// TIA Portal V18 export
TYPE "LGasp_typeRigaProdfromPC"
// stored: IsFailsafeCompliant false
   STRUCT
      piecestodo : DInt;   // Pezzi da fare
      ID : DInt;   // ID riga di produzione
      tipoarticolo : DInt;   // tipo articolo
      info : Struct   // info varie variabili da macchina a macchina
         collo : Int;
         workorder : DInt;
         IDERP : DInt;
      END_STRUCT;
      article : "LGasp_typeArticolo";
   END_STRUCT;
END_TYPE
